{attribute addProperty BoxType "EP5101-0011-0016"}
{attribute addProperty Id "ENC_Status_compactAT %I*ENC_Status_compact_3D346E774860ENC_Control_compactAT %Q*ENC_Control_compact_03701F333240WcStateAT %I*WcState_F855686C1620InfoDataAT %I*InfoData_BC63D37F80100"}
{attribute addProperty CRC "1718053656"}
{attribute addProperty SizeInBites "176"}
{attribute addProperty SizeInBytes "22"}
TYPE EP5101_BA9EF925 :
STRUCT
	{attribute addProperty Name "ENC_Status_compact"}
	ENC_Status_compact : ENC_Status_compact_3D346E77;
	{attribute addProperty Name "ENC_Control_compact"}
	ENC_Control_compact : ENC_Control_compact_03701F33;
	{attribute addProperty Name "WcState"}
	WcState : WcState_F855686C;
	{attribute addProperty Name "InfoData"}
	InfoData : InfoData_BC63D37F;
END_STRUCT
END_TYPE

(* stored: Version 1.2.0.0, ProductVersion 3.1.4024.9
   DUT EP5101_BA9EF925: Id {0ed42874-16b4-41fc-90b2-63d8703ef617} *)
